SYSTEM CODEC_TEST2L (* PUBL/SUBL Test with Derived Data Types *)
  (* Standard: 61499-1ITA; Classification: Communications; Function: Test System *)
  (* Version 1.0, 2007-11-08, JHC, Holobloc Inc, Corrected initialization of matrices. *)
  (* Version 0.9, 2004-06-23, JHC, Rockwell Automation, Deleted MONITOR (not used). *)
  (* Version 0.8, 2004-06-22, JHC, Rockwell Automation, Modified to use IN_MATRIX, OUT_MATRIX. *)
  (* Version 0.7, 2003-12-04, JHC, Rockwell Automation, Removed QI's from PUBL/SUBLs *)
  (* Version 0.6, 2002-03-08, JHC, Rockwell Automation, Added M_IO for MATRIX I/O *)
  (* Version 0.5, 2002-03-06, JHC, Rockwell Automation, Added TEST_MATRIX, single TEST frame *)
  (* Version 0.4, 2001-06-13, JHC, Rockwell Automation, Added applications including TEST_AI16C. *)
  (* Version 0.3, 2001-06-08, JHC, Rockwell Automation, Corrected UDP addresses; changed GUIs to IN_ANY, OUT_ANY *)
  (* Version 0.2, 2001-05-30, JHC, Rockwell Automation, Saved layouts *)
  (* Version 0.1, 2000-05-16, JHC, Rockwell Automation, File type changed to ".sys" *)
  (* Version 0.0, 2000-04-19, JHC, Rockwell Automation *)
  APPLICATION TEST_REAL_VS
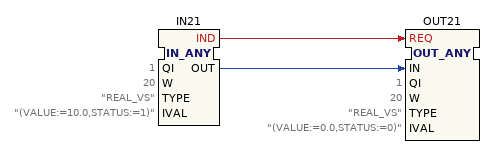
    FBS
      IN21 : IN_ANY(QI := 1, W := 20, TYPE := "REAL_VS", IVAL := "(VALUE:=10.0,STATUS:=1)");
      OUT21 : OUT_ANY(QI := 1, W := 20, TYPE := "REAL_VS", IVAL := "(VALUE:=0.0,STATUS:=0)");
    END_FBS
    EVENT_CONNECTIONS
      IN21.IND TO OUT21.REQ;
    END_CONNECTIONS
    DATA_CONNECTIONS
      IN21.OUT TO OUT21.IN;
    END_CONNECTIONS
  END_APPLICATION
  APPLICATION TEST_ENUMS
    FBS
      IN1 : IN_ENUM(QI := 1, TYPE := "ANALOG_SIGNAL_TYPE");
      IN2 : IN_ENUM(QI := 1, TYPE := "ANALOG_SIGNAL_RANGE");
      OUT1 : OUT_ANY(QI := 1, W := 20, TYPE := "ANALOG_SIGNAL_TYPE");
      OUT2 : OUT_ANY(QI := 1, W := 20, TYPE := "ANALOG_SIGNAL_RANGE");
    END_FBS
    EVENT_CONNECTIONS
      IN1.INITO TO IN2.INIT;
      IN1.IND TO IN2.REQ;
      IN2.IND TO OUT1.REQ;
      OUT1.INITO TO OUT2.INIT;
      OUT1.CNF TO OUT2.REQ;
    END_CONNECTIONS
    DATA_CONNECTIONS
      IN1.OUT TO OUT1.IN;
      IN2.OUT TO OUT2.IN;
    END_CONNECTIONS
  END_APPLICATION
  APPLICATION TEST_FREQ
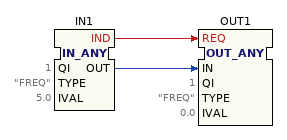
    FBS
      IN1 : IN_ANY(QI := 1, TYPE := "FREQ", IVAL := 5.0);
      OUT1 : OUT_ANY(QI := 1, TYPE := "FREQ", IVAL := 0.0);
    END_FBS
    EVENT_CONNECTIONS
      IN1.IND TO OUT1.REQ;
    END_CONNECTIONS
    DATA_CONNECTIONS
      IN1.OUT TO OUT1.IN;
    END_CONNECTIONS
  END_APPLICATION
  APPLICATION TEST_SUBR
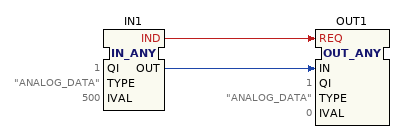
    FBS
      IN1 : IN_ANY(QI := 1, TYPE := "ANALOG_DATA", IVAL := 500);
      OUT1 : OUT_ANY(QI := 1, TYPE := "ANALOG_DATA", IVAL := 0);
    END_FBS
    EVENT_CONNECTIONS
      IN1.IND TO OUT1.REQ;
    END_CONNECTIONS
    DATA_CONNECTIONS
      IN1.OUT TO OUT1.IN;
    END_CONNECTIONS
  END_APPLICATION
  APPLICATION TEST_AI16
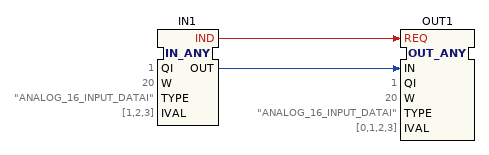
    FBS
      IN1 : IN_ANY(QI := 1, W := 20, TYPE := "ANALOG_16_INPUT_DATAI", IVAL := [1,2,3]);
      OUT1 : OUT_ANY(QI := 1, W := 20, TYPE := "ANALOG_16_INPUT_DATAI", IVAL := [0,1,2,3]);
    END_FBS
    EVENT_CONNECTIONS
      IN1.IND TO OUT1.REQ;
    END_CONNECTIONS
    DATA_CONNECTIONS
      IN1.OUT TO OUT1.IN;
    END_CONNECTIONS
  END_APPLICATION
  APPLICATION TEST_AI16C (* Test ANALOG_16_INPUT_CONFIGURATION *)
    FBS
      IN1 : IN_ANY(QI := 1, W := 20, TYPE := "ANALOG_16_INPUT_CONFIGURATION");
      OUT1 : OUT_ANY(QI := 1, W := 20, TYPE := "ANALOG_16_INPUT_CONFIGURATION");
    END_FBS
    EVENT_CONNECTIONS
      IN1.IND TO OUT1.REQ;
    END_CONNECTIONS
    DATA_CONNECTIONS
      IN1.OUT TO OUT1.IN;
    END_CONNECTIONS
  END_APPLICATION
  APPLICATION TEST_MATRIX
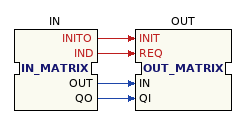
    FBS
      IN : IN_MATRIX;
      OUT : OUT_MATRIX;
    END_FBS
    EVENT_CONNECTIONS
      IN.INITO TO OUT.INIT;
      IN.IND TO OUT.REQ;
    END_CONNECTIONS
    DATA_CONNECTIONS
      IN.OUT TO OUT.IN;
      IN.QO TO OUT.QI;
    END_CONNECTIONS
  END_APPLICATION
  DEVICE TEST : FRAME_DEVICE(BOUNDS := [100,250,800,320], GRID := [4,4])
    RESOURCE SEND_REAL_VS : PANEL_RESOURCE
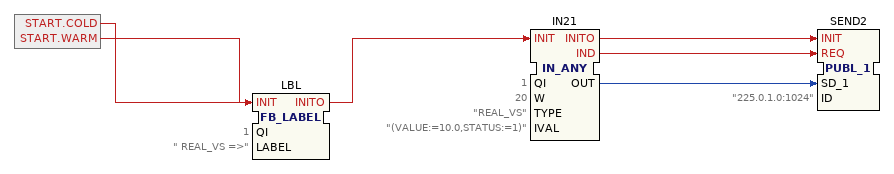
      FBS
        LBL : FB_LABEL(QI := 1, LABEL := " REAL_VS =>");
        IN21 : IN_ANY(QI := 1, W := 20, TYPE := "REAL_VS", IVAL := "(VALUE:=10.0,STATUS:=1)");
        SEND2 : PUBL_1(ID := "225.0.1.0:1024");
      END_FBS
      EVENT_CONNECTIONS
        START.COLD TO LBL.INIT;
        START.WARM TO LBL.INIT;
        LBL.INITO TO IN21.INIT;
        IN21.INITO TO SEND2.INIT;
        IN21.IND TO SEND2.REQ;
      END_CONNECTIONS
      DATA_CONNECTIONS
        IN21.OUT TO SEND2.SD_1;
      END_CONNECTIONS
    END_RESOURCE
    RESOURCE RCV_REAL_VS : PANEL_RESOURCE
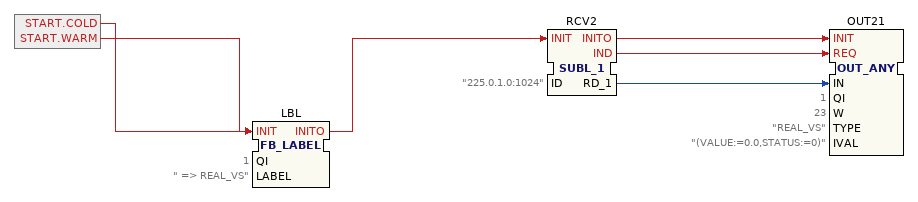
      FBS
        LBL : FB_LABEL(QI := 1, LABEL := " => REAL_VS");
        RCV2 : SUBL_1(ID := "225.0.1.0:1024");
        OUT21 : OUT_ANY(QI := 1, W := 23, TYPE := "REAL_VS", IVAL := "(VALUE:=0.0,STATUS:=0)");
      END_FBS
      EVENT_CONNECTIONS
        START.COLD TO LBL.INIT;
        START.WARM TO LBL.INIT;
        LBL.INITO TO RCV2.INIT;
        RCV2.INITO TO OUT21.INIT;
        RCV2.IND TO OUT21.REQ;
      END_CONNECTIONS
      DATA_CONNECTIONS
        RCV2.RD_1 TO OUT21.IN;
      END_CONNECTIONS
    END_RESOURCE
    RESOURCE SEND_ENUMS : PANEL_RESOURCE
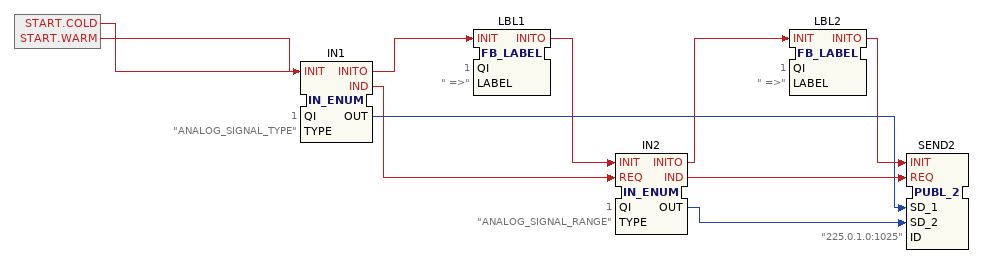
      FBS
        IN1 : IN_ENUM(QI := 1, TYPE := "ANALOG_SIGNAL_TYPE");
        LBL1 : FB_LABEL(QI := 1, LABEL := " =>");
        IN2 : IN_ENUM(QI := 1, TYPE := "ANALOG_SIGNAL_RANGE");
        LBL2 : FB_LABEL(QI := 1, LABEL := " =>");
        SEND2 : PUBL_2(ID := "225.0.1.0:1025");
      END_FBS
      EVENT_CONNECTIONS
        START.COLD TO IN1.INIT;
        START.WARM TO IN1.INIT;
        IN1.INITO TO LBL1.INIT;
        LBL1.INITO TO IN2.INIT;
        IN2.INITO TO LBL2.INIT;
        LBL2.INITO TO SEND2.INIT;
        IN1.IND TO IN2.REQ;
        IN2.IND TO SEND2.REQ;
      END_CONNECTIONS
      DATA_CONNECTIONS
        IN1.OUT TO SEND2.SD_1;
        IN2.OUT TO SEND2.SD_2;
      END_CONNECTIONS
    END_RESOURCE
    RESOURCE RCV_ENUMS : PANEL_RESOURCE
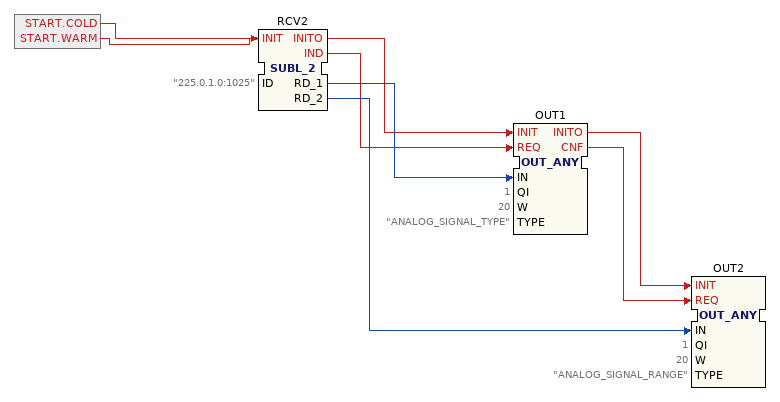
      FBS
        RCV2 : SUBL_2(ID := "225.0.1.0:1025");
        OUT1 : OUT_ANY(QI := 1, W := 20, TYPE := "ANALOG_SIGNAL_TYPE");
        OUT2 : OUT_ANY(QI := 1, W := 20, TYPE := "ANALOG_SIGNAL_RANGE");
      END_FBS
      EVENT_CONNECTIONS
        START.COLD TO RCV2.INIT;
        START.WARM TO RCV2.INIT;
        RCV2.INITO TO OUT1.INIT;
        OUT1.INITO TO OUT2.INIT;
        RCV2.IND TO OUT1.REQ;
        OUT1.CNF TO OUT2.REQ;
      END_CONNECTIONS
      DATA_CONNECTIONS
        RCV2.RD_1 TO OUT1.IN;
        RCV2.RD_2 TO OUT2.IN;
      END_CONNECTIONS
    END_RESOURCE
    RESOURCE SEND_FREQ : PANEL_RESOURCE
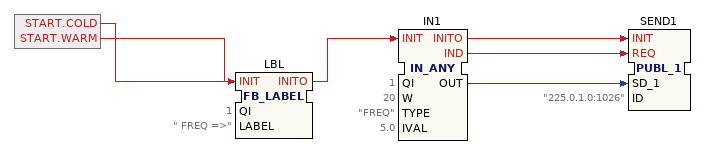
      FBS
        LBL : FB_LABEL(QI := 1, LABEL := " FREQ =>");
        IN1 : IN_ANY(QI := 1, W := 20, TYPE := "FREQ", IVAL := 5.0);
        SEND1 : PUBL_1(ID := "225.0.1.0:1026");
      END_FBS
      EVENT_CONNECTIONS
        START.COLD TO LBL.INIT;
        START.WARM TO LBL.INIT;
        LBL.INITO TO IN1.INIT;
        IN1.INITO TO SEND1.INIT;
        IN1.IND TO SEND1.REQ;
      END_CONNECTIONS
      DATA_CONNECTIONS
        IN1.OUT TO SEND1.SD_1;
      END_CONNECTIONS
    END_RESOURCE
    RESOURCE RCV_FREQ : PANEL_RESOURCE
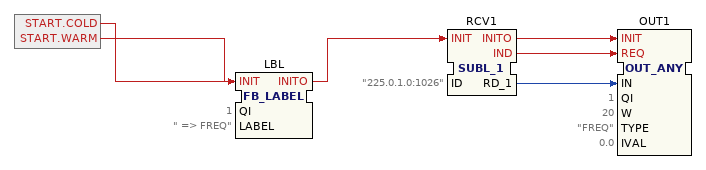
      FBS
        LBL : FB_LABEL(QI := 1, LABEL := " => FREQ");
        RCV1 : SUBL_1(ID := "225.0.1.0:1026");
        OUT1 : OUT_ANY(QI := 1, W := 20, TYPE := "FREQ", IVAL := 0.0);
      END_FBS
      EVENT_CONNECTIONS
        START.COLD TO LBL.INIT;
        START.WARM TO LBL.INIT;
        LBL.INITO TO RCV1.INIT;
        RCV1.INITO TO OUT1.INIT;
        RCV1.IND TO OUT1.REQ;
      END_CONNECTIONS
      DATA_CONNECTIONS
        RCV1.RD_1 TO OUT1.IN;
      END_CONNECTIONS
    END_RESOURCE
    RESOURCE SEND_SUBR : PANEL_RESOURCE
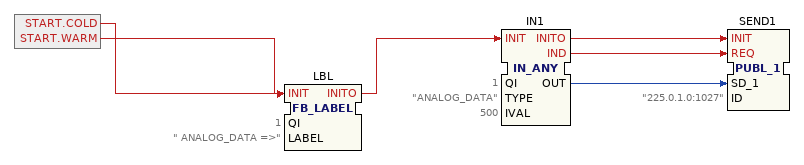
      FBS
        LBL : FB_LABEL(QI := 1, LABEL := " ANALOG_DATA =>");
        IN1 : IN_ANY(QI := 1, TYPE := "ANALOG_DATA", IVAL := 500);
        SEND1 : PUBL_1(ID := "225.0.1.0:1027");
      END_FBS
      EVENT_CONNECTIONS
        START.COLD TO LBL.INIT;
        START.WARM TO LBL.INIT;
        LBL.INITO TO IN1.INIT;
        IN1.INITO TO SEND1.INIT;
        IN1.IND TO SEND1.REQ;
      END_CONNECTIONS
      DATA_CONNECTIONS
        IN1.OUT TO SEND1.SD_1;
      END_CONNECTIONS
    END_RESOURCE
    RESOURCE RCV_SUBR : PANEL_RESOURCE
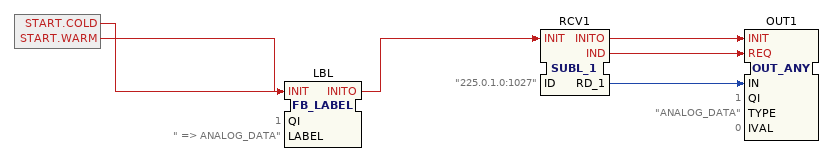
      FBS
        LBL : FB_LABEL(QI := 1, LABEL := " => ANALOG_DATA");
        RCV1 : SUBL_1(ID := "225.0.1.0:1027");
        OUT1 : OUT_ANY(QI := 1, TYPE := "ANALOG_DATA", IVAL := 0);
      END_FBS
      EVENT_CONNECTIONS
        START.COLD TO LBL.INIT;
        START.WARM TO LBL.INIT;
        LBL.INITO TO RCV1.INIT;
        RCV1.INITO TO OUT1.INIT;
        RCV1.IND TO OUT1.REQ;
      END_CONNECTIONS
      DATA_CONNECTIONS
        RCV1.RD_1 TO OUT1.IN;
      END_CONNECTIONS
    END_RESOURCE
    RESOURCE SEND_AI16 : PANEL_RESOURCE
      FBS
        LBL : FB_LABEL(QI := 1, LABEL := " ANALOG_16_INPUT_DATAI =>");
        IN1 : IN_ANY(QI := 1, W := 20, TYPE := "ANALOG_16_INPUT_DATAI", IVAL := [1,2,3]);
        SEND1 : PUBL_1(ID := "225.0.1.0:1028");
      END_FBS
      EVENT_CONNECTIONS
        START.COLD TO LBL.INIT;
        START.WARM TO LBL.INIT;
        LBL.INITO TO IN1.INIT;
        IN1.INITO TO SEND1.INIT;
        IN1.IND TO SEND1.REQ;
      END_CONNECTIONS
      DATA_CONNECTIONS
        IN1.OUT TO SEND1.SD_1;
      END_CONNECTIONS
    END_RESOURCE
    RESOURCE RCV_AI16 : PANEL_RESOURCE
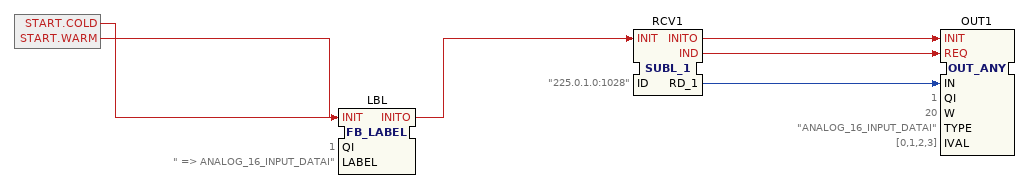
      FBS
        LBL : FB_LABEL(QI := 1, LABEL := " => ANALOG_16_INPUT_DATAI");
        RCV1 : SUBL_1(ID := "225.0.1.0:1028");
        OUT1 : OUT_ANY(QI := 1, W := 20, TYPE := "ANALOG_16_INPUT_DATAI", IVAL := [0,1,2,3]);
      END_FBS
      EVENT_CONNECTIONS
        START.COLD TO LBL.INIT;
        START.WARM TO LBL.INIT;
        LBL.INITO TO RCV1.INIT;
        RCV1.INITO TO OUT1.INIT;
        RCV1.IND TO OUT1.REQ;
      END_CONNECTIONS
      DATA_CONNECTIONS
        RCV1.RD_1 TO OUT1.IN;
      END_CONNECTIONS
    END_RESOURCE
    RESOURCE SEND_AI16C : PANEL_RESOURCE
      FBS
        LBL : FB_LABEL(QI := 1, LABEL := "ANALOG_16_INPUT_... =>");
        IN1 : IN_ANY(QI := 1, W := 20, TYPE := "ANALOG_16_INPUT_CONFIGURATION", IVAL := (SIGNAL_TYPE:=DIFFERENTIAL,FILTER:=50,CHANNEL:=[(RANGE:=UNIPOLAR_10V),(MAX_SCALE:= 100, MIN_SCALE:=0)]));
        SEND1 : PUBL_1(ID := "225.0.1.0:1029");
      END_FBS
      EVENT_CONNECTIONS
        START.COLD TO LBL.INIT;
        START.WARM TO LBL.INIT;
        LBL.INITO TO IN1.INIT;
        IN1.INITO TO SEND1.INIT;
        IN1.IND TO SEND1.REQ;
      END_CONNECTIONS
      DATA_CONNECTIONS
        IN1.OUT TO SEND1.SD_1;
      END_CONNECTIONS
    END_RESOURCE
    RESOURCE RCV_AI16C : PANEL_RESOURCE
      FBS
        LBL : FB_LABEL(QI := 1, LABEL := " => ..._CONFIGURATION");
        RCV1 : SUBL_1(ID := "225.0.1.0:1029");
        OUT1 : OUT_ANY(QI := 1, W := 20, TYPE := "ANALOG_16_INPUT_CONFIGURATION");
      END_FBS
      EVENT_CONNECTIONS
        START.COLD TO LBL.INIT;
        START.WARM TO LBL.INIT;
        LBL.INITO TO RCV1.INIT;
        RCV1.INITO TO OUT1.INIT;
        RCV1.IND TO OUT1.REQ;
      END_CONNECTIONS
      DATA_CONNECTIONS
        RCV1.RD_1 TO OUT1.IN;
      END_CONNECTIONS
    END_RESOURCE
    RESOURCE SEND_MATRIX : PANEL_RESOURCE(ROWS := 1, COLS := 1)
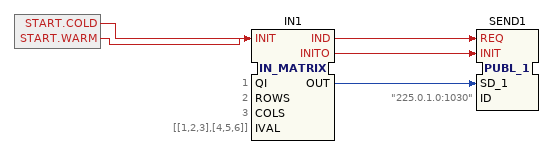
      FBS
        IN1 : IN_MATRIX(QI := 1, ROWS := 2, COLS := 3, IVAL := [[1,2,3],[4,5,6]]);
        SEND1 : PUBL_1(ID := "225.0.1.0:1030");
      END_FBS
      EVENT_CONNECTIONS
        START.COLD TO IN1.INIT;
        START.WARM TO IN1.INIT;
        IN1.IND TO SEND1.REQ;
        IN1.INITO TO SEND1.INIT;
      END_CONNECTIONS
      DATA_CONNECTIONS
        IN1.OUT TO SEND1.SD_1;
      END_CONNECTIONS
    END_RESOURCE
    RESOURCE RCV_MATRIX : PANEL_RESOURCE(ROWS := 1, COLS := 1)
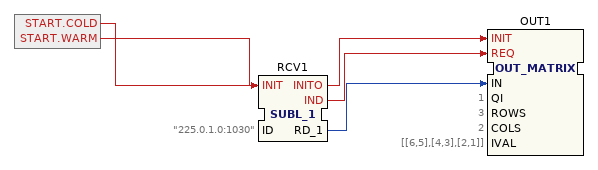
      FBS
        RCV1 : SUBL_1(ID := "225.0.1.0:1030");
        OUT1 : OUT_MATRIX(QI := 1, ROWS := 3, COLS := 2, IVAL := [[6,5],[4,3],[2,1]]);
      END_FBS
      EVENT_CONNECTIONS
        START.COLD TO RCV1.INIT;
        START.WARM TO RCV1.INIT;
        RCV1.INITO TO OUT1.INIT;
        RCV1.IND TO OUT1.REQ;
      END_CONNECTIONS
      DATA_CONNECTIONS
        RCV1.RD_1 TO OUT1.IN;
      END_CONNECTIONS
    END_RESOURCE
  END_DEVICE
END_SYSTEM
